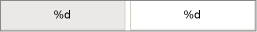
VISUALIZATION VISU_ConfigUDINTEntry  // 257x32
VAR_IN_OUT
    active : UDINT;
    editable : UDINT;
END_VAR
    Textfield (0,0 125x30), "%d", text variable: active, input disabled if: TRUE
    Textfield (130,0 125x30), "%d", text variable: editable, colour toggle: editable <> active
        OnMouseClick: write the text variable via Default
END_VISUALIZATION

(* stored: Version 1.1.0.1, ProductVersion 3.1.0.36
   Visu VISU_ConfigUDINTEntry: Id {5a638977-193f-4087-9df9-f359eb5405ed} *)
